(* PLC project MQTT, OpenPLC MQTT 1.0, author OpenPLC Lib Writter *)
(* stored: creationDateTime 2023-04-26T04:54:00, modificationDateTime 2023-04-26T04:54:00 *)

(* Setups RS-485 interface to send and receive data through serial wire when CONNECT is triggered. If setup is successful, SUCCESS is set to TRUE. Interface transfer BAUDRATE and STOPBITS can be configured. Also there is an opportunity to control terminal resistors via ENABLE_TERMINAL_RESISTORS flag. *)
FUNCTION_BLOCK RS485_CONNECT
  VAR_INPUT
    CONNECT : BOOL;
    ENABLE_TERMINAL_RESISTORS : BOOL := TRUE;
    BAUDRATE : UDINT := 115200;
    STOPBITS : USINT := 1;
  END_VAR
  VAR_OUTPUT
    SUCCESS : BOOL;
  END_VAR

            SUCCESS := FALSE;
          
END_FUNCTION_BLOCK

(* Sends a MESSAGE through RS-485 interface. If the sending was successful then SUCCESS is set to TRUE. If receiving has already been started then the message can't be sent. (max MESSAGE ARRAY size is 128 bytes, indexes start from 0). *)
FUNCTION_BLOCK RS485_SEND_BYTES
  VAR_INPUT
    SEND : BOOL;
    MESSAGE_SIZE : USINT;
    MESSAGE : ARRAY[0..127] OF BYTE;
  END_VAR
  VAR_OUTPUT
    SUCCESS : BOOL;
  END_VAR

            SUCCESS := FALSE;
          
END_FUNCTION_BLOCK

(* Starts receiving from RS485 ciclically, saves every RECEIVE_PACKET_SIZE bytes into packet. If the starting was successful then SUCCESS is set to TRUE. The packet size can't be more than 128 bytes. *)
FUNCTION_BLOCK RS485_START_RECEIVING
  VAR_INPUT
    START : BOOL;
    RECEIVE_PACKET_SIZE : USINT;
  END_VAR
  VAR_OUTPUT
    SUCCESS : BOOL;
  END_VAR

            SUCCESS := FALSE;
          
END_FUNCTION_BLOCK

(* Disconnects from RS485 interface. If the disconnection was successfull then SUCCESS is set to TRUE. *)
FUNCTION_BLOCK RS485_DISCONNECT
  VAR_INPUT
    DISCONNECT : BOOL;
  END_VAR
  VAR_OUTPUT
    SUCCESS : BOOL;
  END_VAR

            SUCCESS := FALSE;
          
END_FUNCTION_BLOCK

(* Gets next received packet, returns packet itself and its size. If there isn't any packet then RECEIVED_PACKET_SIZE will be equal to zero. *)
FUNCTION_BLOCK RS485_GET_NEXT_RECEIVED_PACKET
  VAR_INPUT
    GET : BOOL;
  END_VAR
  VAR_OUTPUT
    RECEIVED_PACKET_SIZE : USINT;
    RECEIVED_PACKET : ARRAY[0..127] OF BYTE;
  END_VAR

            RECEIVED_PACKET_SIZE := 0;
          
END_FUNCTION_BLOCK

(* Stops receiving data from RS485 interface. If the stopping was successful then SUCCESS is set to TRUE. *)
FUNCTION_BLOCK RS485_STOP_RECEIVING
  VAR_INPUT
    STOP : BOOL;
  END_VAR
  VAR_OUTPUT
    SUCCESS : BOOL;
  END_VAR

            SUCCESS := FALSE;
          
END_FUNCTION_BLOCK
